FUNCTION_BLOCK FB_ExecutorBase EXTENDS FB_CyclicFB IMPLEMENTS I_MachiningExecutor, I_BB8Specification
VAR
    // Zmienne sekwencyjne 
    nStep           : INT;
    iCurrentSegment : INT;
    StepTimer       : TON;
    _bBusy          : BOOL;
    _bDone          : BOOL;
    _bError         : BOOL;
    _uErrorID       : UDINT;

    // --- ZMIENNE WSPÓLNE DLA WSZYSTKICH EXECUTORÓW
    _AxisX          : SPT_Motion_Control.I_BasicAxis;
    _AxisY          : SPT_Motion_Control.I_BasicAxis;
    _AxisZ          : SPT_Motion_Control.I_BasicAxis;
    _Cylinder       : I_Cylinder;                     
    _RecipeBuilder  : I_RecipeBuilder;
    _Config         : REFERENCE TO ST_GantryXYZ_Config;
END_VAR

METHOD Abort
_bBusy := FALSE;
_bDone := FALSE;
nStep := 0;
iCurrentSegment := 1;
StepTimer(IN := FALSE);
END_METHOD

PROPERTY AxisX : I_BasicAxis
GET
AxisX := _AxisX;
END_GET
SET
_AxisX := AxisX;
END_SET
END_PROPERTY

PROPERTY AxisY : I_BasicAxis
GET
AxisY := _AxisY;
END_GET
SET
_AxisY := AxisY;
END_SET
END_PROPERTY

PROPERTY AxisZ : I_BasicAxis
GET
AxisZ := _AxisZ;
END_GET
SET
_AxisZ := AxisZ;
END_SET
END_PROPERTY

PROPERTY Busy : BOOL
GET
Busy := _bBusy;
END_GET
END_PROPERTY

PROPERTY Config : REFERENCE TO ST_GantryXYZ_Config
GET
Config REF= _Config;
END_GET
SET
_Config REF= Config;
END_SET
END_PROPERTY

METHOD PUBLIC  CyclicLogic
VAR_INPUT
END_VAR
END_METHOD

PROPERTY Cylinder : I_Cylinder
GET
Cylinder := _Cylinder;
END_GET
SET
_Cylinder := Cylinder;
END_SET
END_PROPERTY

PROPERTY Done : BOOL
GET
Done := _bDone;
END_GET
END_PROPERTY

PROPERTY Error : BOOL
GET
Error := _bError;
END_GET
END_PROPERTY


PROPERTY ErrorID : UDINT
GET
ErrorID := _uErrorID;
END_GET
END_PROPERTY

METHOD Execute : BOOL
IF _bBusy THEN RETURN; END_IF

_bBusy    := TRUE;
_bDone    := FALSE;
_bError   := FALSE;
_uErrorID := 0;
nStep     := 5; 
Execute   := TRUE;
END_METHOD

PROPERTY RecipeBuilder : I_RecipeBuilder
GET
RecipeBuilder := _RecipeBuilder;
END_GET
SET
_RecipeBuilder := RecipeBuilder;
END_SET
END_PROPERTY

END_FUNCTION_BLOCK

(* stored: Version 1.1.0.1, ProductVersion 3.1.4024.15
   POU FB_ExecutorBase: Id {0cbe7356-7a09-405e-9aff-39065bb1c2f0}, SpecialFunc None
   Method Abort: Id {6635fc89-ad71-4ff9-bc14-3af14ce8aecc}
   Property AxisX: Id {bf7bf1e8-4628-46ee-9a7f-8b243677db34}
   Get Get: Id {d93144b5-dd29-483a-8b76-9038e49c9a6d}
   Set Set: Id {7ab3348b-b4bb-4d6b-bd39-8185e257a35e}
   Property AxisY: Id {d6d2cedb-0eda-4e75-a191-4d8ce3a9bbf4}
   Get Get: Id {3b91612c-9793-4f68-8ba4-cfcfaf6d0685}
   Set Set: Id {cefe518b-6ed4-4e66-9928-cc421068c6b9}
   Property AxisZ: Id {411509dc-9082-4584-89ca-2ff1afd18787}
   Get Get: Id {3ef8d70c-0902-4da9-8ae9-200f5cfec13c}
   Set Set: Id {fbb69cdf-dc2f-457b-88ac-db5f43779a82}
   Property Busy: Id {59913f19-c467-40c0-a679-c67212e49f90}
   Get Get: Id {5507dde5-0c97-489e-a157-38e3094c1db6}
   Property Config: Id {d4eaeb02-3324-4dfb-bb21-b43618bd8a51}
   Get Get: Id {b1b19422-708f-4729-8a80-0ec5c4e56462}
   Set Set: Id {855da8aa-c381-42d4-945c-30bcec476610}
   Method CyclicLogic: Id {668c6d27-30c6-490b-b139-36714103a9b4}
   Property Cylinder: Id {0546bd86-401b-41c0-a683-bbe302146fdd}
   Get Get: Id {622de191-a52d-4efd-af87-b0787b5827c2}
   Set Set: Id {f831b18a-1816-415a-82f6-5aeacd4161b5}
   Property Done: Id {2d95981e-5455-46ef-8af6-2891542aa2dc}
   Get Get: Id {d1a57449-624d-4917-966a-8665e0388821}
   Property Error: Id {8c239f0b-1fc4-4c24-a95e-da15dbc5c2fc}
   Get Get: Id {9b4d655e-598b-457a-88d2-81afba639fe2}
   Property ErrorID: Id {dbbab504-dbb1-4393-938e-b24e98188e14}
   Get Get: Id {83105c2a-ef7b-4470-ad8e-857d462980fa}
   Method Execute: Id {c37f539b-c1c9-4761-b6a7-a09dc0c33fb5}
   Property RecipeBuilder: Id {cbbaad3b-7e73-402c-b55d-1c46460bfd77}
   Get Get: Id {ee8216eb-1e0d-45e3-8dfd-22bbcbfa2526}
   Set Set: Id {1d93da46-a542-4ef2-b525-3599ad0c4f6e} *)
